TEXTLIST tlPML_Commands
  0 = 'PMLCommand_Undefined'
  1 = 'PMLCommand_Reset'
  2 = 'PMLCommand_Start'
  3 = 'PMLCommand_Stop'
  4 = 'PMLCommand_Hold'
  5 = 'PMLCommand_Unhold'
  6 = 'PMLCommand_Suspend'
  7 = 'PMLCommand_Unsuspend'
  8 = 'PMLCommand_Abort'
  9 = 'PMLCommand_Clear'
   = ''
END_TEXTLIST

(* stored: Version 1.1.0.1, ProductVersion 3.1.4024.11
   TextList tlPML_Commands: Id {466d29a5-104c-4c12-a7b2-792958dc834a} *)
